PROGRAM MAIN
VAR
	nCounter	: UINT;
	fbCountTime	: TON := (PT:=T#1S);
END_VAR

IF _TaskInfo[GETCURTASKINDEXEX()].FirstCycle THEN
	F_Log(E_LogLevel.eInfo, 'SPS Task gestartet.');
END_IF

fbCountTime(IN:=NOT fbCountTime.Q);
IF fbCountTime.Q THEN
	nCounter := nCounter + 1;
	F_LogA1(E_LogLevel.eDebug, 'Zähler geändert, neuer Wert {0}', nCounter);
END_IF

PRG_TaskLog.Call();

END_PROGRAM

(* stored: Version 1.1.0.1, ProductVersion 3.1.4024.0
   POU MAIN: Id {df1e3a16-6581-4c31-b5b6-204a618c6fef}, SpecialFunc None *)
